KUKA KRL program: ps_ltc_geo_x1.src, ps_ltc_geo_x1.dat

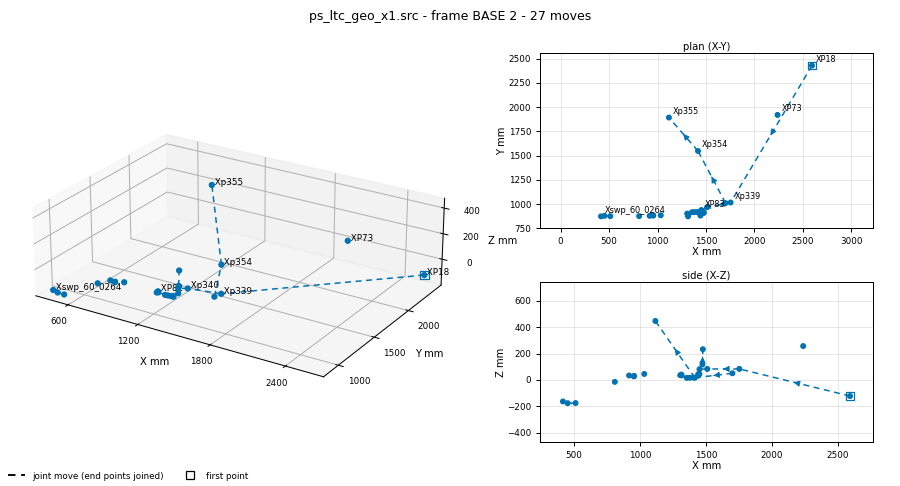
[picture p0: tool path of ps_ltc_geo_x1.src in frame BASE 2, 27 of 45 moves have a stored position in this frame; points joined in program order, loops and branches not executed]
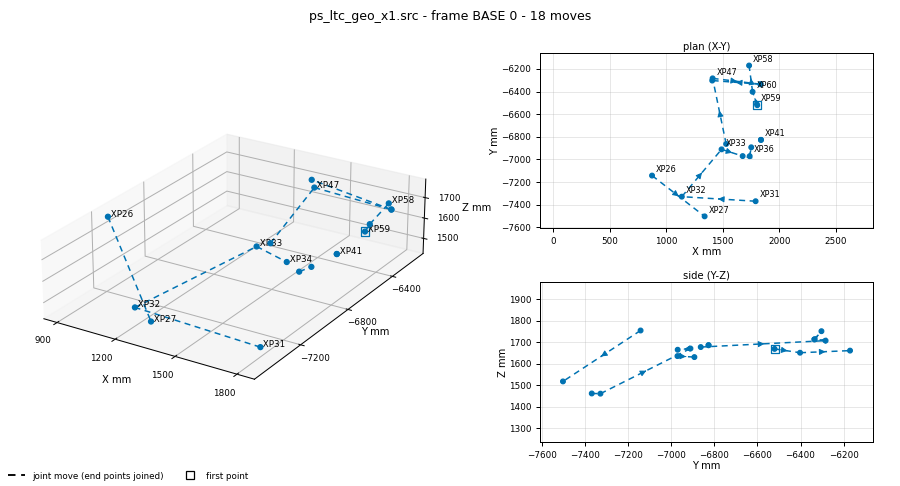
[picture p1: tool path of ps_ltc_geo_x1.src in frame BASE 0, 18 of 45 moves have a stored position in this frame; points joined in program order, loops and branches not executed]
--- ps_ltc_geo_x1.src ---
&ACCESS RVO2
&REL 14
&COMMENT Solda GUN X1 geometria
&PARAM DISKPATH = KRC:\R1\Program\SOLDA LTC
DEF ps_ltc_geo_x1( )

;FOLD INI
  ;FOLD BASISTECH INI
    GLOBAL INTERRUPT DECL 3 WHEN $STOPMESS==TRUE DO IR_STOPM ( )
    INTERRUPT ON 3
    BAS (#INITMOV,0 )
  ;ENDFOLD (BASISTECH INI)
;FOLD SPOTTECH INI
USERSPOT(#INIT)
;ENDFOLD (SPOTTECH INI)
;FOLD GRIPPERTECH INI
USER_GRP(0,DUMMY,DUMMY,GDEFAULT)
;ENDFOLD (GRIPPERTECH INI)
  ;FOLD USER INI
    ;Make your modifications here

  ;ENDFOLD (USER INI)
;ENDFOLD (INI)

; Caracterização dos meios de produção:
; Versão Atual:
; 01/05/2013 12:00 Name: P13.050-R2 CHANGES: Solda Geometria
; Pinça X1, Accelo

chk_w1_wechs_ok ( )    ; CHECK TOOL X1

if MaxStandMenge (4) then
MaxStandmengeErreicht (4)
endif

IF (NOT(GHOST())) THEN
if FraesAnf(4) then
e_fraes1 ()
endif
ENDIF

;FOLD PTP P18 CONT Vel=100 % PDAT100 Tool[1]:Gun X1 Base[2]:Accelo;%{PE}%R 8.2.20,%MKUKATPBASIS,%CMOVE,%VPTP,%P 1:PTP, 2:P18, 3:C_DIS, 5:100, 7:PDAT100
$BWDSTART=FALSE
PDAT_ACT=PPDAT100
FDAT_ACT=FP18
BAS(#PTP_PARAMS,100)
PTP XP18 C_DIS
;ENDFOLD
;FOLD PTP p339 CONT Vel=100 % PDAT30 Tool[1]:Gun X1 Base[2]:Accelo;%{PE}%R 8.2.20,%MKUKATPBASIS,%CMOVE,%VPTP,%P 1:PTP, 2:p339, 3:C_DIS, 5:100, 7:PDAT30
$BWDSTART=FALSE
PDAT_ACT=PPDAT30
FDAT_ACT=Fp339
BAS(#PTP_PARAMS,100)
PTP Xp339 C_DIS
;ENDFOLD
;FOLD PTP p340 CONT Vel=100 % PDAT31 Tool[1]:Gun X1 Base[2]:Accelo;%{PE}%R 8.2.20,%MKUKATPBASIS,%CMOVE,%VPTP,%P 1:PTP, 2:p340, 3:C_DIS, 5:100, 7:PDAT31
$BWDSTART=FALSE
PDAT_ACT=PPDAT31
FDAT_ACT=Fp340
BAS(#PTP_PARAMS,100)
PTP Xp340 C_DIS
;ENDFOLD

;FOLD OUT 3339 'R2 solicita lib. para soldar geometria' State=TRUE ;%{PE}%R 8.2.20,%MKUKATPBASIS,%COUT,%VOUTX,%P 2:3339, 3:R2 solicita lib. para soldar geometria, 5:TRUE, 6:
$OUT[3339]=TRUE
;ENDFOLD
;FOLD WAIT FOR ( IN 3339 'R2 aguarda lib. Soldar geometria' );%{PE}%R 8.2.20,%MKUKATPBASIS,%CEXT_WAIT_FOR,%VEXT_WAIT_FOR,%P 2:, 4:, 5:$IN, 6:3339, 7:R2 aguarda lib.  Soldar geometria, 9:
WAIT FOR  ( $IN[3339] )
;ENDFOLD
;FOLD OUT 3339 'R2 solicita lib. para soldar geometria' State=FALSE ;%{PE}%R 8.2.20,%MKUKATPBASIS,%COUT,%VOUTX,%P 2:3339, 3:R2 solicita lib. para soldar geometria, 5:FALSE, 6:
$OUT[3339]=FALSE
;ENDFOLD
;FOLD OUT 3348 'Fora area GEOBOX' State=FALSE ;%{PE}%R 8.2.20,%MKUKATPBASIS,%COUT,%VOUTX,%P 2:3348, 3:Fora area GEOBOX, 5:FALSE, 6:
$OUT[3348]=FALSE
;ENDFOLD

;FOLD Collision.Monitoring_AREA_1_On ;%{PE}%MKUKATPUSER
COLLSTOP( 7, 1 ) ;not Interrupt-Controlled
;ENDFOLD

;FOLD PTP p341 CONT Vel=100 % PDAT91 Tool[1]:Gun X1 Base[2]:Accelo;%{PE}%R 8.2.20,%MKUKATPBASIS,%CMOVE,%VPTP,%P 1:PTP, 2:p341, 3:C_DIS, 5:100, 7:PDAT91
$BWDSTART=FALSE
PDAT_ACT=PPDAT91
FDAT_ACT=Fp341
BAS(#PTP_PARAMS,100)
PTP Xp341 C_DIS
;ENDFOLD
;FOLD PTP P83 CONT Vel=100 % PDAT166 Tool[1]:Gun X1 Base[2]:Accelo;%{PE}%R 8.2.20,%MKUKATPBASIS,%CMOVE,%VPTP,%P 1:PTP, 2:P83, 3:C_DIS, 5:100, 7:PDAT166
$BWDSTART=FALSE
PDAT_ACT=PPDAT166
FDAT_ACT=FP83
BAS(#PTP_PARAMS,100)
PTP XP83 C_DIS
;ENDFOLD

; SP0328
;FOLD PTP swp_60_0328 PDAT104 SPOT Gun=4 RETR CLS PGNO1=100 ACTIVE=1 Tool[1]:Gun X1 Base[2]:Accelo;%{PE}%R 8.2.2,%MKUKATPSPOT,%CSPOT,%VPTP,%P 1:PTP, 2:swp_60_0328, 3:, 5:100, 7:PDAT104, 10:4, 12:#FIRST, 14:#CLO, 16:181, 18:1, 20:0, 22:0, 24:1, 25:NORMAL
$BWDSTART=FALSE
PDAT_ACT=PPDAT104
FDAT_ACT=Fswp_60_0328
BAS(#PTP_PARAMS,PPDAT104.VEL)
S_ACT.GUN=4
S_ACT.PAIR=SDEFAULT.PAIR
S_ACT.RETR=#CLO
S_ACT.CLO_TM=1
S_ACT.PGNO1=100
S_ACT.PGNO2=SDEFAULT.PGNO2
S_ACT.PRESS1=SDEFAULT.PRESS1
S_ACT.PRESS2=SDEFAULT.PRESS2
S_READY=FALSE
PTP Xswp_60_0328
USERSPOT(#SPOT, S_ACT)
WAIT FOR S_READY
;ENDFOLD

; SP0326
;FOLD PTP swp_60_0326 PDAT157 SPOT Gun=4 RETR OPN PGNO1=132 ACTIVE=1 Tool[1]:Gun X1 Base[2]:Accelo;%{PE}%R 8.2.2,%MKUKATPSPOT,%CSPOT,%VPTP,%P 1:PTP, 2:swp_60_0326, 3:, 5:100, 7:PDAT157, 10:4, 12:#FIRST, 14:#OPN, 16:213, 18:1, 20:0, 22:0, 24:1, 25:NORMAL
$BWDSTART=FALSE
PDAT_ACT=PPDAT157
FDAT_ACT=Fswp_60_0326
BAS(#PTP_PARAMS,PPDAT157.VEL)
S_ACT.GUN=4
S_ACT.PAIR=SDEFAULT.PAIR
S_ACT.RETR=#OPN
S_ACT.CLO_TM=1
S_ACT.PGNO1=132
S_ACT.PGNO2=SDEFAULT.PGNO2
S_ACT.PRESS1=SDEFAULT.PRESS1
S_ACT.PRESS2=SDEFAULT.PRESS2
S_READY=FALSE
PTP Xswp_60_0326
USERSPOT(#SPOT, S_ACT)
WAIT FOR S_READY
;ENDFOLD

; SP0324
;FOLD PTP swp_60_0324 PDAT158 SPOT Gun=4 RETR CLS PGNO1=121 ACTIVE=1 Tool[1]:Gun X1 Base[2]:Accelo;%{PE}%R 8.2.2,%MKUKATPSPOT,%CSPOT,%VPTP,%P 1:PTP, 2:swp_60_0324, 3:, 5:100, 7:PDAT158, 10:4, 12:#FIRST, 14:#CLO, 16:202, 18:1, 20:0, 22:0, 24:1, 25:NORMAL
$BWDSTART=FALSE
PDAT_ACT=PPDAT158
FDAT_ACT=Fswp_60_0324
BAS(#PTP_PARAMS,PPDAT158.VEL)
S_ACT.GUN=4
S_ACT.PAIR=SDEFAULT.PAIR
S_ACT.RETR=#CLO
S_ACT.CLO_TM=1
S_ACT.PGNO1=121
S_ACT.PGNO2=SDEFAULT.PGNO2
S_ACT.PRESS1=SDEFAULT.PRESS1
S_ACT.PRESS2=SDEFAULT.PRESS2
S_READY=FALSE
PTP Xswp_60_0324
USERSPOT(#SPOT, S_ACT)
WAIT FOR S_READY
;ENDFOLD

; SP0322
;FOLD PTP swp_60_0322 PDAT159 SPOT Gun=4 RETR CLS PGNO1=133 ACTIVE=1 Tool[1]:Gun X1 Base[2]:Accelo;%{PE}%R 8.2.2,%MKUKATPSPOT,%CSPOT,%VPTP,%P 1:PTP, 2:swp_60_0322, 3:, 5:100, 7:PDAT159, 10:4, 12:#FIRST, 14:#CLO, 16:214, 18:1, 20:0, 22:0, 24:1, 25:NORMAL
$BWDSTART=FALSE
PDAT_ACT=PPDAT159
FDAT_ACT=Fswp_60_0322
BAS(#PTP_PARAMS,PPDAT159.VEL)
S_ACT.GUN=4
S_ACT.PAIR=SDEFAULT.PAIR
S_ACT.RETR=#CLO
S_ACT.CLO_TM=1
S_ACT.PGNO1=133
S_ACT.PGNO2=SDEFAULT.PGNO2
S_ACT.PRESS1=SDEFAULT.PRESS1
S_ACT.PRESS2=SDEFAULT.PRESS2
S_READY=FALSE
PTP Xswp_60_0322
USERSPOT(#SPOT, S_ACT)
WAIT FOR S_READY
;ENDFOLD

; SP0320
;FOLD PTP swp_60_0320 PDAT160 SPOT Gun=4 RETR OPN PGNO1=134 ACTIVE=1 Tool[1]:Gun X1 Base[2]:Accelo;%{PE}%R 8.2.2,%MKUKATPSPOT,%CSPOT,%VPTP,%P 1:PTP, 2:swp_60_0320, 3:, 5:100, 7:PDAT160, 10:4, 12:#FIRST, 14:#OPN, 16:215, 18:1, 20:0, 22:0, 24:1, 25:NORMAL
$BWDSTART=FALSE
PDAT_ACT=PPDAT160
FDAT_ACT=Fswp_60_0320
BAS(#PTP_PARAMS,PPDAT160.VEL)
S_ACT.GUN=4
S_ACT.PAIR=SDEFAULT.PAIR
S_ACT.RETR=#OPN
S_ACT.CLO_TM=1
S_ACT.PGNO1=134
S_ACT.PGNO2=SDEFAULT.PGNO2
S_ACT.PRESS1=SDEFAULT.PRESS1
S_ACT.PRESS2=SDEFAULT.PRESS2
S_READY=FALSE
PTP Xswp_60_0320
USERSPOT(#SPOT, S_ACT)
WAIT FOR S_READY
;ENDFOLD

; SP0318
;FOLD PTP swp_60_0318 PDAT161 SPOT Gun=4 RETR OPN PGNO1=122 ACTIVE=1 Tool[1]:Gun X1 Base[2]:Accelo;%{PE}%R 8.2.2,%MKUKATPSPOT,%CSPOT,%VPTP,%P 1:PTP, 2:swp_60_0318, 3:, 5:100, 7:PDAT161, 10:4, 12:#FIRST, 14:#OPN, 16:203, 18:1, 20:0, 22:0, 24:1, 25:NORMAL
$BWDSTART=FALSE
PDAT_ACT=PPDAT161
FDAT_ACT=Fswp_60_0318
BAS(#PTP_PARAMS,PPDAT161.VEL)
S_ACT.GUN=4
S_ACT.PAIR=SDEFAULT.PAIR
S_ACT.RETR=#OPN
S_ACT.CLO_TM=1
S_ACT.PGNO1=122
S_ACT.PGNO2=SDEFAULT.PGNO2
S_ACT.PRESS1=SDEFAULT.PRESS1
S_ACT.PRESS2=SDEFAULT.PRESS2
S_READY=FALSE
PTP Xswp_60_0318
USERSPOT(#SPOT, S_ACT)
WAIT FOR S_READY
;ENDFOLD

; SP0316
;FOLD PTP swp_60_0316 PDAT167 SPOT Gun=4 RETR OPN PGNO1=135 ACTIVE=1 Tool[1]:Gun X1 Base[2]:Accelo;%{PE}%R 8.2.2,%MKUKATPSPOT,%CSPOT,%VPTP,%P 1:PTP, 2:swp_60_0316, 3:, 5:100, 7:PDAT167, 10:4, 12:#FIRST, 14:#OPN, 16:216, 18:1, 20:0, 22:0, 24:1, 25:NORMAL
$BWDSTART=FALSE
PDAT_ACT=PPDAT167
FDAT_ACT=Fswp_60_0316
BAS(#PTP_PARAMS,PPDAT167.VEL)
S_ACT.GUN=4
S_ACT.PAIR=SDEFAULT.PAIR
S_ACT.RETR=#OPN
S_ACT.CLO_TM=1
S_ACT.PGNO1=135
S_ACT.PGNO2=SDEFAULT.PGNO2
S_ACT.PRESS1=SDEFAULT.PRESS1
S_ACT.PRESS2=SDEFAULT.PRESS2
S_READY=FALSE
PTP Xswp_60_0316
USERSPOT(#SPOT, S_ACT)
WAIT FOR S_READY
;ENDFOLD

;FOLD PTP P82 CONT Vel=100 % PDAT165 Tool[1]:Gun X1 Base[2]:Accelo;%{PE}%R 8.2.20,%MKUKATPBASIS,%CMOVE,%VPTP,%P 1:PTP, 2:P82, 3:C_DIS, 5:100, 7:PDAT165
$BWDSTART=FALSE
PDAT_ACT=PPDAT165
FDAT_ACT=FP82
BAS(#PTP_PARAMS,100)
PTP XP82 C_DIS
;ENDFOLD
;FOLD PTP P59 CONT Vel=100 % PDAT141 Tool[1]:Gun X1 Base[2]:Accelo;%{PE}%R 8.2.20,%MKUKATPBASIS,%CMOVE,%VPTP,%P 1:PTP, 2:P59, 3:C_DIS, 5:100, 7:PDAT141
$BWDSTART=FALSE
PDAT_ACT=PPDAT141
FDAT_ACT=FP59
BAS(#PTP_PARAMS,100)
PTP XP59 C_DIS
;ENDFOLD
;FOLD PTP P60 CONT Vel=100 % PDAT142 Tool[1]:Gun X1 Base[2]:Accelo;%{PE}%R 8.2.20,%MKUKATPBASIS,%CMOVE,%VPTP,%P 1:PTP, 2:P60, 3:C_DIS, 5:100, 7:PDAT142
$BWDSTART=FALSE
PDAT_ACT=PPDAT142
FDAT_ACT=FP60
BAS(#PTP_PARAMS,100)
PTP XP60 C_DIS
;ENDFOLD
;FOLD PTP P58 CONT Vel=100 % PDAT140 Tool[1]:Gun X1 Base[2]:Accelo;%{PE}%R 8.2.20,%MKUKATPBASIS,%CMOVE,%VPTP,%P 1:PTP, 2:P58, 3:C_DIS, 5:100, 7:PDAT140
$BWDSTART=FALSE
PDAT_ACT=PPDAT140
FDAT_ACT=FP58
BAS(#PTP_PARAMS,100)
PTP XP58 C_DIS
;ENDFOLD
;FOLD PTP P10 Vel=100 % PDAT92 Tool[1]:Gun X1 Base[2]:Accelo;%{PE}%R 8.2.20,%MKUKATPBASIS,%CMOVE,%VPTP,%P 1:PTP, 2:P10, 3:, 5:100, 7:PDAT92
$BWDSTART=FALSE
PDAT_ACT=PPDAT92
FDAT_ACT=FP10
BAS(#PTP_PARAMS,100)
PTP XP10
;ENDFOLD

;FOLD Collision.Monitoring_AREA_1_Off . ;%{PE}%MKUKATPUSER
COLLSTOP( 7, 2+0 )
;ENDFOLD
;FOLD Collision.Monitoring_AREA_2_On ;%{PE}%MKUKATPUSER
COLLSTOP( 8, 1 ) ;not Interrupt-Controlled
;ENDFOLD
;FOLD Collision.Monitoring_4_On ;%{PE}%MKUKATPUSER
COLLSTOP( 4, 1 ) ;Interrupt-Controlled
;ENDFOLD

;FOLD PTP p354 CONT Vel=100 % PDAT44 Tool[1]:Gun X1 Base[2]:Accelo;%{PE}%R 8.2.20,%MKUKATPBASIS,%CMOVE,%VPTP,%P 1:PTP, 2:p354, 3:C_DIS, 5:100, 7:PDAT44
$BWDSTART=FALSE
PDAT_ACT=PPDAT44
FDAT_ACT=Fp354
BAS(#PTP_PARAMS,100)
PTP Xp354 C_DIS
;ENDFOLD
;FOLD PTP p355 CONT Vel=100 % PDAT45 Tool[1]:Gun X1 Base[2]:Accelo;%{PE}%R 8.2.20,%MKUKATPBASIS,%CMOVE,%VPTP,%P 1:PTP, 2:p355, 3:C_DIS, 5:100, 7:PDAT45
$BWDSTART=FALSE
PDAT_ACT=PPDAT45
FDAT_ACT=Fp355
BAS(#PTP_PARAMS,100)
PTP Xp355 C_DIS
;ENDFOLD
;FOLD PTP P26 CONT Vel=100 % PDAT108 Tool[1]:Gun X1 Base[2]:Accelo;%{PE}%R 8.2.20,%MKUKATPBASIS,%CMOVE,%VPTP,%P 1:PTP, 2:P26, 3:C_DIS, 5:100, 7:PDAT108
$BWDSTART=FALSE
PDAT_ACT=PPDAT108
FDAT_ACT=FP26
BAS(#PTP_PARAMS,100)
PTP XP26 C_DIS
;ENDFOLD
;FOLD PTP P27 CONT Vel=100 % PDAT109 Tool[1]:Gun X1 Base[2]:Accelo;%{PE}%R 8.2.20,%MKUKATPBASIS,%CMOVE,%VPTP,%P 1:PTP, 2:P27, 3:C_DIS, 5:100, 7:PDAT109
$BWDSTART=FALSE
PDAT_ACT=PPDAT109
FDAT_ACT=FP27
BAS(#PTP_PARAMS,100)
PTP XP27 C_DIS
;ENDFOLD

; SP0264
;FOLD PTP swp_60_0264 PDAT151 SPOT Gun=4 RETR CLS PGNO1=109 ACTIVE=1 Tool[1]:Gun X1 Base[2]:Accelo;%{PE}%R 8.2.2,%MKUKATPSPOT,%CSPOT,%VPTP,%P 1:PTP, 2:swp_60_0264, 3:, 5:100, 7:PDAT151, 10:4, 12:#FIRST, 14:#CLO, 16:190, 18:1, 20:0, 22:0, 24:1, 25:NORMAL
$BWDSTART=FALSE
PDAT_ACT=PPDAT151
FDAT_ACT=Fswp_60_0264
BAS(#PTP_PARAMS,PPDAT151.VEL)
S_ACT.GUN=4
S_ACT.PAIR=SDEFAULT.PAIR
S_ACT.RETR=#CLO
S_ACT.CLO_TM=1
S_ACT.PGNO1=109
S_ACT.PGNO2=SDEFAULT.PGNO2
S_ACT.PRESS1=SDEFAULT.PRESS1
S_ACT.PRESS2=SDEFAULT.PRESS2
S_READY=FALSE
PTP Xswp_60_0264
USERSPOT(#SPOT, S_ACT)
WAIT FOR S_READY
;ENDFOLD

;FOLD PTP P84 CONT Vel=100 % PDAT168 Tool[1]:Gun X1 Base[2]:Accelo;%{PE}%R 8.2.20,%MKUKATPBASIS,%CMOVE,%VPTP,%P 1:PTP, 2:P84, 3:C_DIS, 5:100, 7:PDAT168
$BWDSTART=FALSE
PDAT_ACT=PPDAT168
FDAT_ACT=FP84
BAS(#PTP_PARAMS,100)
PTP XP84 C_DIS
;ENDFOLD

; SP0268
;FOLD PTP swp_60_0268 PDAT150 SPOT Gun=4 RETR OPN PGNO1=108 ACTIVE=1 Tool[1]:Gun X1 Base[2]:Accelo;%{PE}%R 8.2.2,%MKUKATPSPOT,%CSPOT,%VPTP,%P 1:PTP, 2:swp_60_0268, 3:, 5:100, 7:PDAT150, 10:4, 12:#FIRST, 14:#OPN, 16:189, 18:1, 20:0, 22:0, 24:1, 25:NORMAL
$BWDSTART=FALSE
PDAT_ACT=PPDAT150
FDAT_ACT=Fswp_60_0268
BAS(#PTP_PARAMS,PPDAT150.VEL)
S_ACT.GUN=4
S_ACT.PAIR=SDEFAULT.PAIR
S_ACT.RETR=#OPN
S_ACT.CLO_TM=1
S_ACT.PGNO1=108
S_ACT.PGNO2=SDEFAULT.PGNO2
S_ACT.PRESS1=SDEFAULT.PRESS1
S_ACT.PRESS2=SDEFAULT.PRESS2
S_READY=FALSE
PTP Xswp_60_0268
USERSPOT(#SPOT, S_ACT)
WAIT FOR S_READY
;ENDFOLD

;FOLD PTP P31 CONT Vel=100 % PDAT113 Tool[1]:Gun X1 Base[2]:Accelo;%{PE}%R 8.2.20,%MKUKATPBASIS,%CMOVE,%VPTP,%P 1:PTP, 2:P31, 3:C_DIS, 5:100, 7:PDAT113
$BWDSTART=FALSE
PDAT_ACT=PPDAT113
FDAT_ACT=FP31
BAS(#PTP_PARAMS,100)
PTP XP31 C_DIS
;ENDFOLD
;FOLD PTP P32 CONT Vel=100 % PDAT114 Tool[1]:Gun X1 Base[2]:Accelo;%{PE}%R 8.2.20,%MKUKATPBASIS,%CMOVE,%VPTP,%P 1:PTP, 2:P32, 3:C_DIS, 5:100, 7:PDAT114
$BWDSTART=FALSE
PDAT_ACT=PPDAT114
FDAT_ACT=FP32
BAS(#PTP_PARAMS,100)
PTP XP32 C_DIS
;ENDFOLD
;FOLD PTP P33 CONT Vel=100 % PDAT115 Tool[1]:Gun X1 Base[2]:Accelo;%{PE}%R 8.2.20,%MKUKATPBASIS,%CMOVE,%VPTP,%P 1:PTP, 2:P33, 3:C_DIS, 5:100, 7:PDAT115
$BWDSTART=FALSE
PDAT_ACT=PPDAT115
FDAT_ACT=FP33
BAS(#PTP_PARAMS,100)
PTP XP33 C_DIS
;ENDFOLD
;FOLD PTP P34 CONT Vel=100 % PDAT116 Tool[1]:Gun X1 Base[2]:Accelo;%{PE}%R 8.2.20,%MKUKATPBASIS,%CMOVE,%VPTP,%P 1:PTP, 2:P34, 3:C_DIS, 5:100, 7:PDAT116
$BWDSTART=FALSE
PDAT_ACT=PPDAT116
FDAT_ACT=FP34
BAS(#PTP_PARAMS,100)
PTP XP34 C_DIS
;ENDFOLD

; SP0284
;FOLD PTP swp_60_0284 PDAT143 SPOT Gun=4 RETR OPN PGNO1=107 ACTIVE=1 Tool[1]:Gun X1 Base[2]:Accelo;%{PE}%R 8.2.2,%MKUKATPSPOT,%CSPOT,%VPTP,%P 1:PTP, 2:swp_60_0284, 3:, 5:100, 7:PDAT143, 10:4, 12:#FIRST, 14:#OPN, 16:188, 18:1, 20:0, 22:0, 24:1, 25:NORMAL
$BWDSTART=FALSE
PDAT_ACT=PPDAT143
FDAT_ACT=Fswp_60_0284
BAS(#PTP_PARAMS,PPDAT143.VEL)
S_ACT.GUN=4
S_ACT.PAIR=SDEFAULT.PAIR
S_ACT.RETR=#OPN
S_ACT.CLO_TM=1
S_ACT.PGNO1=107
S_ACT.PGNO2=SDEFAULT.PGNO2
S_ACT.PRESS1=SDEFAULT.PRESS1
S_ACT.PRESS2=SDEFAULT.PRESS2
S_READY=FALSE
PTP Xswp_60_0284
USERSPOT(#SPOT, S_ACT)
WAIT FOR S_READY
;ENDFOLD

;FOLD PTP P36 CONT Vel=100 % PDAT118 Tool[1]:Gun X1 Base[2]:Accelo;%{PE}%R 8.2.20,%MKUKATPBASIS,%CMOVE,%VPTP,%P 1:PTP, 2:P36, 3:C_DIS, 5:100, 7:PDAT118
$BWDSTART=FALSE
PDAT_ACT=PPDAT118
FDAT_ACT=FP36
BAS(#PTP_PARAMS,100)
PTP XP36 C_DIS
;ENDFOLD
;FOLD PTP P37 CONT Vel=100 % PDAT119 Tool[1]:Gun X1 Base[2]:Accelo;%{PE}%R 8.2.20,%MKUKATPBASIS,%CMOVE,%VPTP,%P 1:PTP, 2:P37, 3:C_DIS, 5:100, 7:PDAT119
$BWDSTART=FALSE
PDAT_ACT=PPDAT119
FDAT_ACT=FP37
BAS(#PTP_PARAMS,100)
PTP XP37 C_DIS
;ENDFOLD
;FOLD PTP P62 PDAT144 RETR CLS Gun=4 Tool[1]:Gun X1 Base[2]:Accelo;%{PE}%R 8.2.2,%MKUKATPSPOT,%CRETR,%VPTP,%P 1:PTP, 2:P62, 3:, 5:100, 7:PDAT144, 9:#CLO, 11:4, 13:#FIRST
$BWDSTART=FALSE
PDAT_ACT=PPDAT144
FDAT_ACT=FP62
BAS(#PTP_PARAMS,PPDAT144.VEL)
S_ACT.GUN=4
S_ACT.PAIR=#FIRST
S_ACT.RETR=#CLO
S_READY=FALSE
PTP XP62
USERSPOT(#RETR, S_ACT)
WAIT FOR S_READY
;ENDFOLD

; SP0290
;FOLD PTP swp_60_0290 PDAT145 SPOT Gun=4 RETR CLS PGNO1=106 ACTIVE=1 Tool[1]:Gun X1 Base[2]:Accelo;%{PE}%R 8.2.2,%MKUKATPSPOT,%CSPOT,%VPTP,%P 1:PTP, 2:swp_60_0290, 3:, 5:100, 7:PDAT145, 10:4, 12:#FIRST, 14:#CLO, 16:187, 18:1, 20:0, 22:0, 24:1, 25:NORMAL
$BWDSTART=FALSE
PDAT_ACT=PPDAT145
FDAT_ACT=Fswp_60_0290
BAS(#PTP_PARAMS,PPDAT145.VEL)
S_ACT.GUN=4
S_ACT.PAIR=SDEFAULT.PAIR
S_ACT.RETR=#CLO
S_ACT.CLO_TM=1
S_ACT.PGNO1=106
S_ACT.PGNO2=SDEFAULT.PGNO2
S_ACT.PRESS1=SDEFAULT.PRESS1
S_ACT.PRESS2=SDEFAULT.PRESS2
S_READY=FALSE
PTP Xswp_60_0290
USERSPOT(#SPOT, S_ACT)
WAIT FOR S_READY
;ENDFOLD

;FOLD PTP P41 CONT Vel=100 % PDAT123 Tool[1]:Gun X1 Base[2]:Accelo;%{PE}%R 8.2.20,%MKUKATPBASIS,%CMOVE,%VPTP,%P 1:PTP, 2:P41, 3:C_DIS, 5:100, 7:PDAT123
$BWDSTART=FALSE
PDAT_ACT=PPDAT123
FDAT_ACT=FP41
BAS(#PTP_PARAMS,100)
PTP XP41 C_DIS
;ENDFOLD

; SP0296
;FOLD PTP swp_60_0296 PDAT147 SPOT Gun=4 RETR CLS PGNO1=105 ACTIVE=1 Tool[1]:Gun X1 Base[2]:Accelo;%{PE}%R 8.2.2,%MKUKATPSPOT,%CSPOT,%VPTP,%P 1:PTP, 2:swp_60_0296, 3:, 5:100, 7:PDAT147, 10:4, 12:#FIRST, 14:#CLO, 16:186, 18:1, 20:0, 22:0, 24:1, 25:NORMAL
$BWDSTART=FALSE
PDAT_ACT=PPDAT147
FDAT_ACT=Fswp_60_0296
BAS(#PTP_PARAMS,PPDAT147.VEL)
S_ACT.GUN=4
S_ACT.PAIR=SDEFAULT.PAIR
S_ACT.RETR=#CLO
S_ACT.CLO_TM=1
S_ACT.PGNO1=105
S_ACT.PGNO2=SDEFAULT.PGNO2
S_ACT.PRESS1=SDEFAULT.PRESS1
S_ACT.PRESS2=SDEFAULT.PRESS2
S_READY=FALSE
PTP Xswp_60_0296
USERSPOT(#SPOT, S_ACT)
WAIT FOR S_READY
;ENDFOLD

;FOLD Collision.Monitoring_AREA_2_Off . ;%{PE}%MKUKATPUSER
COLLSTOP( 8, 2+0 )
;ENDFOLD
;FOLD Collision.Monitoring_AREA_3_On ;%{PE}%MKUKATPUSER
COLLSTOP( 9, 1 ) ;not Interrupt-Controlled
;ENDFOLD

;FOLD PTP P43 CONT Vel=100 % PDAT125 Tool[1]:Gun X1 Base[2]:Accelo;%{PE}%R 8.2.20,%MKUKATPBASIS,%CMOVE,%VPTP,%P 1:PTP, 2:P43, 3:C_DIS, 5:100, 7:PDAT125
$BWDSTART=FALSE
PDAT_ACT=PPDAT125
FDAT_ACT=FP43
BAS(#PTP_PARAMS,100)
PTP XP43 C_DIS
;ENDFOLD
;FOLD PTP P71 PDAT153 RETR OPN Gun=4 Tool[1]:Gun X1 Base[2]:Accelo;%{PE}%R 8.2.2,%MKUKATPSPOT,%CRETR,%VPTP,%P 1:PTP, 2:P71, 3:, 5:100, 7:PDAT153, 9:#OPN, 11:4, 13:#FIRST
$BWDSTART=FALSE
PDAT_ACT=PPDAT153
FDAT_ACT=FP71
BAS(#PTP_PARAMS,PPDAT153.VEL)
S_ACT.GUN=4
S_ACT.PAIR=#FIRST
S_ACT.RETR=#OPN
S_READY=FALSE
PTP XP71
USERSPOT(#RETR, S_ACT)
WAIT FOR S_READY
;ENDFOLD
;FOLD PTP P45 CONT Vel=100 % PDAT127 Tool[1]:Gun X1 Base[2]:Accelo;%{PE}%R 8.2.20,%MKUKATPBASIS,%CMOVE,%VPTP,%P 1:PTP, 2:P45, 3:C_DIS, 5:100, 7:PDAT127
$BWDSTART=FALSE
PDAT_ACT=PPDAT127
FDAT_ACT=FP45
BAS(#PTP_PARAMS,100)
PTP XP45 C_DIS
;ENDFOLD
;FOLD PTP P47 CONT Vel=100 % PDAT129 Tool[1]:Gun X1 Base[2]:Accelo;%{PE}%R 8.2.20,%MKUKATPBASIS,%CMOVE,%VPTP,%P 1:PTP, 2:P47, 3:C_DIS, 5:100, 7:PDAT129
$BWDSTART=FALSE
PDAT_ACT=PPDAT129
FDAT_ACT=FP47
BAS(#PTP_PARAMS,100)
PTP XP47 C_DIS
;ENDFOLD
;FOLD PTP P48 CONT Vel=100 % PDAT130 Tool[1]:Gun X1 Base[2]:Accelo;%{PE}%R 8.2.20,%MKUKATPBASIS,%CMOVE,%VPTP,%P 1:PTP, 2:P48, 3:C_DIS, 5:100, 7:PDAT130
$BWDSTART=FALSE
PDAT_ACT=PPDAT130
FDAT_ACT=FP48
BAS(#PTP_PARAMS,100)
PTP XP48 C_DIS
;ENDFOLD

; SP0350
;FOLD PTP swp_60_0350 PDAT148 SPOT Gun=4 RETR CLS PGNO1=104 ACTIVE=1 Tool[1]:Gun X1 Base[2]:Accelo;%{PE}%R 8.2.2,%MKUKATPSPOT,%CSPOT,%VPTP,%P 1:PTP, 2:swp_60_0350, 3:, 5:100, 7:PDAT148, 10:4, 12:#FIRST, 14:#CLO, 16:185, 18:1, 20:0, 22:0, 24:1, 25:NORMAL
$BWDSTART=FALSE
PDAT_ACT=PPDAT148
FDAT_ACT=Fswp_60_0350
BAS(#PTP_PARAMS,PPDAT148.VEL)
S_ACT.GUN=4
S_ACT.PAIR=SDEFAULT.PAIR
S_ACT.RETR=#CLO
S_ACT.CLO_TM=1
S_ACT.PGNO1=104
S_ACT.PGNO2=SDEFAULT.PGNO2
S_ACT.PRESS1=SDEFAULT.PRESS1
S_ACT.PRESS2=SDEFAULT.PRESS2
S_READY=FALSE
PTP Xswp_60_0350
USERSPOT(#SPOT, S_ACT)
WAIT FOR S_READY
;ENDFOLD

; SP0356
;FOLD PTP swp_60_0356 PDAT149 SPOT Gun=4 RETR OPN PGNO1=103 ACTIVE=1 Tool[1]:Gun X1 Base[2]:Accelo;%{PE}%R 8.2.2,%MKUKATPSPOT,%CSPOT,%VPTP,%P 1:PTP, 2:swp_60_0356, 3:, 5:100, 7:PDAT149, 10:4, 12:#FIRST, 14:#OPN, 16:184, 18:1, 20:0, 22:0, 24:1, 25:NORMAL
$BWDSTART=FALSE
PDAT_ACT=PPDAT149
FDAT_ACT=Fswp_60_0356
BAS(#PTP_PARAMS,PPDAT149.VEL)
S_ACT.GUN=4
S_ACT.PAIR=SDEFAULT.PAIR
S_ACT.RETR=#OPN
S_ACT.CLO_TM=1
S_ACT.PGNO1=103
S_ACT.PGNO2=SDEFAULT.PGNO2
S_ACT.PRESS1=SDEFAULT.PRESS1
S_ACT.PRESS2=SDEFAULT.PRESS2
S_READY=FALSE
PTP Xswp_60_0356
USERSPOT(#SPOT, S_ACT)
WAIT FOR S_READY
;ENDFOLD

;FOLD PTP P52 CONT Vel=100 % PDAT134 Tool[1]:Gun X1 Base[2]:Accelo;%{PE}%R 8.2.20,%MKUKATPBASIS,%CMOVE,%VPTP,%P 1:PTP, 2:P52, 3:C_DIS, 5:100, 7:PDAT134
$BWDSTART=FALSE
PDAT_ACT=PPDAT134
FDAT_ACT=FP52
BAS(#PTP_PARAMS,100)
PTP XP52 C_DIS
;ENDFOLD
;FOLD PTP P53 CONT Vel=100 % PDAT135 Tool[1]:Gun X1 Base[2]:Accelo;%{PE}%R 8.2.20,%MKUKATPBASIS,%CMOVE,%VPTP,%P 1:PTP, 2:P53, 3:C_DIS, 5:100, 7:PDAT135
$BWDSTART=FALSE
PDAT_ACT=PPDAT135
FDAT_ACT=FP53
BAS(#PTP_PARAMS,100)
PTP XP53 C_DIS
;ENDFOLD
;FOLD PTP P73 Vel=100 % PDAT155 Tool[1]:Gun X1 Base[2]:Accelo;%{PE}%R 8.2.20,%MKUKATPBASIS,%CMOVE,%VPTP,%P 1:PTP, 2:P73, 3:, 5:100, 7:PDAT155
$BWDSTART=FALSE
PDAT_ACT=PPDAT155
FDAT_ACT=FP73
BAS(#PTP_PARAMS,100)
PTP XP73
;ENDFOLD

;FOLD Collision.Monitoring_4_Off . ;%{PE}%MKUKATPUSER
COLLSTOP( 4, 2+0 )
;ENDFOLD
;FOLD Collision.Monitoring_AREA_3_Off . ;%{PE}%MKUKATPUSER
COLLSTOP( 9, 2+0 )
;ENDFOLD

;FOLD OUT 3348 'Fora area GEOBOX' State=TRUE ;%{PE}%R 8.2.20,%MKUKATPBASIS,%COUT,%VOUTX,%P 2:3348, 3:Fora area GEOBOX, 5:TRUE, 6:
$OUT[3348]=TRUE
;ENDFOLD

IF (NOT(GHOST())) THEN
if FraesAnf(4) then
f_fraes1 ()
endif
ENDIF

END

--- ps_ltc_geo_x1.dat ---
&ACCESS RVO2
&REL 14
&COMMENT Solda GUN X1 geometria
&PARAM DISKPATH = KRC:\R1\Program\SOLDA LTC
DEFDAT  ps_ltc_geo_x1
;FOLD EXTERNAL DECLARATIONS;%{PE}%MKUKATPBASIS,%CEXT,%VCOMMON,%P
;FOLD GRIPPERTECH EXT
EXT  H50 (INT  :IN,INT  :IN,INT  :IN,GRP_TYP  :IN )
;ENDFOLD (GRIPPERTECH EXT)
;FOLD SPOTTECH EXT
EXT  USERSPOT (S_COMMAND  :IN,SPOT_TYPE  :IN )
;ENDFOLD (SPOTTECH EXT)
;FOLD BASISTECH EXT;%{PE}%MKUKATPBASIS,%CEXT,%VEXT,%P
EXT  BAS (BAS_COMMAND  :IN,REAL  :IN )
DECL INT SUCCESS
;ENDFOLD (BASISTECH EXT)
;FOLD USER EXT;%{E}%MKUKATPUSER,%CEXT,%VEXT,%P
;Make your modifications here

;ENDFOLD (USER EXT)
;ENDFOLD (EXTERNAL DECLARATIONS)

;# ============ START PATH : swp_p13050r2_ltc_geo_x1 =============
DECL FDAT Fswp_60_0326={TOOL_NO 1,BASE_NO 2,IPO_FRAME #BASE,POINT2[] " ",TQ_STATE FALSE}
DECL SPOT_TYPE SS_OLP1={GUN 1,PAIR #FIRST,RETR #OPN,CLO_TM 0,PGNO1 1,PRESS1 1.0,PGNO2 0,PRESS2 0.0}
DECL E6POS Xswp_60_0326={X 1440.89099,Y 894.045471,Z 31.5168095,A -159.997894,B -3.0173409,C -140.140106,S 2,T 35,E1 -4617.46387,E2 0.0,E3 0.0,E4 0.0,E5 0.0,E6 0.0}
DECL FDAT Fswp_60_0322={TOOL_NO 1,BASE_NO 2,IPO_FRAME #BASE,POINT2[] " "}
DECL SPOT_TYPE SS_OLP2={GUN 1,PAIR #FIRST,RETR #OPN,CLO_TM 0,PGNO1 1,PRESS1 1.0,PGNO2 0,PRESS2 0.0}
DECL E6POS Xswp_60_0322={X 1379.50696,Y 917.822388,Z 16.3037205,A -171.276505,B -1.12520099,C -145.708496,S 2,T 35,E1 -4617.46094,E2 0.0,E3 0.0,E4 0.0,E5 0.0,E6 0.0}
DECL FDAT Fswp_60_0318={TOOL_NO 1,BASE_NO 2,IPO_FRAME #BASE,POINT2[] " "}
DECL SPOT_TYPE SS_OLP3={GUN 1,PAIR #FIRST,RETR #OPN,CLO_TM 0,PGNO1 1,PRESS1 1.0,PGNO2 0,PRESS2 0.0}
DECL E6POS Xswp_60_0318={X 1316.23206,Y 893.451721,Z 34.1688995,A -171.866196,B -2.02005601,C -146.172501,S 2,T 35,E1 -4617.52979,E2 0.0,E3 0.0,E4 0.0,E5 0.0,E6 0.0}
DECL FDAT Fswp_60_0356={TOOL_NO 1,BASE_NO 2,IPO_FRAME #BASE,POINT2[] " "}
DECL SPOT_TYPE SS_OLP4={GUN 1,PAIR #FIRST,RETR #OPN,CLO_TM 0,PGNO1 1,PRESS1 1.0,PGNO2 0,PRESS2 0.0}
DECL E6POS Xswp_60_0356={X 1477.68201,Y 913.010681,Z 232.539505,A -91.0726166,B -4.99526501,C 89.5052872,S 6,T 51,E1 -4829.7959,E2 0.0,E3 0.0,E4 0.0,E5 0.0,E6 0.0}
DECL FDAT Fswp_60_0350={TOOL_NO 1,BASE_NO 2,IPO_FRAME #BASE,POINT2[] " "}
DECL SPOT_TYPE SS_OLP5={GUN 1,PAIR #FIRST,RETR #OPN,CLO_TM 0,PGNO1 1,PRESS1 1.0,PGNO2 0,PRESS2 0.0}
DECL E6POS Xswp_60_0350={X 1474.26501,Y 909.548706,Z 116.354202,A -91.1325912,B 4.90854406,C 89.584198,S 6,T 51,E1 -4829.7959,E2 0.0,E3 0.0,E4 0.0,E5 0.0,E6 0.0}
DECL FDAT Fswp_60_0296={TOOL_NO 1,BASE_NO 2,IPO_FRAME #BASE,POINT2[] " "}
DECL SPOT_TYPE SS_OLP6={GUN 1,PAIR #FIRST,RETR #OPN,CLO_TM 0,PGNO1 1,PRESS1 1.0,PGNO2 0,PRESS2 0.0}
DECL E6POS Xswp_60_0296={X 1033.53198,Y 884.917114,Z 45.0556412,A -90.2147217,B 19.7881393,C 15.1591501,S 6,T 19,E1 -4845.0249,E2 0.0,E3 0.0,E4 0.0,E5 0.0,E6 0.0}
DECL FDAT Fswp_60_0290={TOOL_NO 1,BASE_NO 2,IPO_FRAME #BASE,POINT2[] " "}
DECL SPOT_TYPE SS_OLP7={GUN 1,PAIR #FIRST,RETR #OPN,CLO_TM 0,PGNO1 1,PRESS1 1.0,PGNO2 0,PRESS2 0.0}
DECL E6POS Xswp_60_0290={X 918.688782,Y 879.437805,Z 33.3725395,A -96.8630524,B 14.4618196,C 10.1200705,S 6,T 19,E1 -4845.01807,E2 0.0,E3 0.0,E4 0.0,E5 0.0,E6 0.0}
DECL FDAT Fswp_60_0284={TOOL_NO 1,BASE_NO 2,IPO_FRAME #BASE,POINT2[] " "}
DECL SPOT_TYPE SS_OLP8={GUN 1,PAIR #FIRST,RETR #OPN,CLO_TM 0,PGNO1 1,PRESS1 1.0,PGNO2 0,PRESS2 0.0}
DECL E6POS Xswp_60_0284={X 810.263184,Y 876.497681,Z -14.9003096,A -101.040604,B 20.5212498,C 26.0307407,S 6,T 19,E1 -4845.02393,E2 0.0,E3 0.0,E4 0.0,E5 0.0,E6 0.0}
DECL FDAT Fswp_60_0268={TOOL_NO 1,BASE_NO 2,IPO_FRAME #BASE,POINT2[] " "}
DECL SPOT_TYPE SS_OLP9={GUN 1,PAIR #FIRST,RETR #OPN,CLO_TM 0,PGNO1 1,PRESS1 1.0,PGNO2 0,PRESS2 0.0}
DECL E6POS Xswp_60_0268={X 512.70282,Y 875.895813,Z -175.678207,A -80.5816193,B 5.79682779,C 5.26112223,S 6,T 19,E1 -5459.71387,E2 0.0,E3 0.0,E4 0.0,E5 0.0,E6 0.0}
DECL FDAT Fswp_60_0264={TOOL_NO 1,BASE_NO 2,IPO_FRAME #BASE,POINT2[] " "}
DECL SPOT_TYPE SS_OLP10={GUN 1,PAIR #FIRST,RETR #OPN,CLO_TM 0,PGNO1 1,PRESS1 1.0,PGNO2 0,PRESS2 0.0}
DECL E6POS Xswp_60_0264={X 417.230286,Y 874.02771,Z -163.492096,A -83.0655136,B 11.3301601,C -19.7582703,S 6,T 19,E1 -5459.74023,E2 0.0,E3 0.0,E4 0.0,E5 0.0,E6 0.0}
DECL BASIS_SUGG_T LAST_BASIS={POINT1[] "P84                     ",POINT2[] "P84                     ",CP_PARAMS[] "CPDAT0                  ",PTP_PARAMS[] "PDAT168                 ",CONT[] "C_DIS                   ",CP_VEL[] "2.0                     ",PTP_VEL[] "100                     ",SPL_NAME[] "S0                      "}
DECL SPOT_SUGG_T LAST_SPOT={GUN[] "4                       ",RETR_CMD[] "#OPN                    ",CHOISE[] "#FIRST                  ",CLO_TM[] "1                       ",PGNO1[] "203                     ",PRESS1[] "0                       ",PGNO2[] "1                       ",PRESS2[] "0                       ",SPOT_PARAMS[] "NORMAL                  "}
DECL E6POS XP339={X 1754.13196,Y 1016.74298,Z 83.1492615,A -164.185501,B 18.5443897,C -158.434204,S 2,T 35,E1 -4458.23779,E2 0.0,E3 0.0,E4 0.0,E5 0.0,E6 0.0}
DECL FDAT Fp339={TOOL_NO 1,BASE_NO 2,IPO_FRAME #BASE,POINT2[] " ",TQ_STATE FALSE}
DECL PDAT PPDAT30={VEL 100.0,ACC 100.0,APO_DIST 100.0,APO_MODE #CDIS}
DECL E6POS XP340={X 1511.08801,Y 967.887085,Z 82.8026428,A -169.680405,B 7.87629414,C -159.822693,S 2,T 35,E1 -4617.45313,E2 0.0,E3 0.0,E4 0.0,E5 0.0,E6 0.0}
DECL FDAT Fp340={TOOL_NO 1,BASE_NO 2,IPO_FRAME #BASE,POINT2[] " ",TQ_STATE FALSE}
DECL PDAT PPDAT31={VEL 100.0,ACC 100.0,APO_DIST 100.0,APO_MODE #CDIS}
DECL E6POS XP341={X 1451.83398,Y 937.507507,Z 81.1336823,A -171.963394,B 1.64496303,C -160.012405,S 2,T 35,E1 -4617.45313,E2 0.0,E3 0.0,E4 0.0,E5 0.0,E6 0.0}
DECL FDAT Fp341={TOOL_NO 1,BASE_NO 2,IPO_FRAME #BASE,POINT2[] " ",TQ_STATE FALSE}
DECL E6POS XP354={X 1417.54895,Y 1548.25305,Z 16.3868809,A -170.275406,B 20.6585407,C -155.272598,S 2,T 35,E1 -4617.31299,E2 0.0,E3 0.0,E4 0.0,E5 0.0,E6 0.0}
DECL FDAT Fp354={TOOL_NO 1,BASE_NO 2,IPO_FRAME #BASE,POINT2[] " ",TQ_STATE FALSE}
DECL PDAT PPDAT44={VEL 100.0,ACC 100.0,APO_DIST 100.0,APO_MODE #CDIS}
DECL E6POS XP355={X 1117.578,Y 1893.255,Z 446.7435,A -149.1931,B 7.65658712,C -137.427094,S 6,T 51,E1 -4617.31299,E2 0.0,E3 0.0,E4 0.0,E5 0.0,E6 0.0}
DECL FDAT Fp355={TOOL_NO 1,BASE_NO 2,IPO_FRAME #BASE,POINT2[] " ",TQ_STATE FALSE}
DECL PDAT PPDAT45={VEL 100.0,ACC 100.0,APO_DIST 100.0,APO_MODE #CDIS}
DECL PDAT PPDAT91={VEL 100.0,ACC 100.0,APO_DIST 20.0,APO_MODE #CDIS}
DECL PDAT PPDAT92={VEL 100.0,ACC 100.0,APO_DIST 100.0,APO_MODE #CDIS}
DECL E6POS XP10={X 1701.64502,Y 1010.94202,Z 50.3210602,A -171.141296,B 15.6092701,C -169.974899,S 2,T 35,E1 -4617.31299,E2 0.0,E3 0.0,E4 0.0,E5 0.0,E6 0.0}
DECL FDAT FP10={TOOL_NO 1,BASE_NO 2,IPO_FRAME #BASE,POINT2[] " ",TQ_STATE FALSE}
DECL PDAT PPDAT100={VEL 100.0,ACC 100.0,APO_DIST 100.0,APO_MODE #CDIS}
DECL E6POS XP18={X 2593.28198,Y 2429.84009,Z -122.263496,A -172.544495,B 61.4785881,C 178.740707,S 2,T 35,E1 -3217.95093,E2 0.0,E3 0.0,E4 0.0,E5 0.0,E6 0.0}
DECL FDAT FP18={TOOL_NO 1,BASE_NO 2,IPO_FRAME #BASE,POINT2[] " ",TQ_STATE FALSE}
DECL PDAT PPDAT104={VEL 100.0,ACC 100.0,APO_DIST 100.0,APO_MODE #CDIS}
DECL E6POS XP26={X 875.52887,Y -7142.63721,Z 1754.10303,A -42.8865509,B 20.2833996,C 87.7021866,S 6,T 50,E1 -4807.50391,E2 0.0,E3 0.0,E4 0.0,E5 0.0,E6 0.0}
DECL FDAT FP26={TOOL_NO 1,BASE_NO 0,IPO_FRAME #BASE,POINT2[] " ",TQ_STATE FALSE}
DECL PDAT PPDAT108={VEL 100.0,ACC 100.0,APO_DIST 100.0,APO_MODE #CDIS}
DECL E6POS XP27={X 1340.20398,Y -7503.00586,Z 1517.61804,A -19.7759609,B 19.0676498,C -7.15892315,S 6,T 18,E1 -5125.43994,E2 0.0,E3 0.0,E4 0.0,E5 0.0,E6 0.0}
DECL FDAT FP27={TOOL_NO 1,BASE_NO 0,IPO_FRAME #BASE,POINT2[] " ",TQ_STATE FALSE}
DECL PDAT PPDAT109={VEL 100.0,ACC 100.0,APO_DIST 100.0,APO_MODE #CDIS}
DECL E6POS XP31={X 1790.88599,Y -7369.36914,Z 1461.67297,A 3.54338598,B 6.05099392,C 5.29669189,S 6,T 19,E1 -5459.73877,E2 0.0,E3 0.0,E4 0.0,E5 0.0,E6 0.0}
DECL FDAT FP31={TOOL_NO 1,BASE_NO 0,IPO_FRAME #BASE,POINT2[] " ",TQ_STATE FALSE}
DECL PDAT PPDAT113={VEL 100.0,ACC 100.0,APO_DIST 100.0,APO_MODE #CDIS}
DECL E6POS XP32={X 1138.55005,Y -7329.03516,Z 1460.82703,A -24.8452702,B 10.6812496,C 4.63611889,S 6,T 18,E1 -4941.47217,E2 0.0,E3 0.0,E4 0.0,E5 0.0,E6 0.0}
DECL FDAT FP32={TOOL_NO 1,BASE_NO 0,IPO_FRAME #BASE,POINT2[] " ",TQ_STATE FALSE}
DECL PDAT PPDAT114={VEL 100.0,ACC 100.0,APO_DIST 100.0,APO_MODE #CDIS}
DECL E6POS XP33={X 1489.85596,Y -6911.00586,Z 1670.39795,A -11.8927603,B 15.9203901,C 14.7493296,S 6,T 19,E1 -4941.48291,E2 0.0,E3 0.0,E4 0.0,E5 0.0,E6 0.0}
DECL FDAT FP33={TOOL_NO 1,BASE_NO 0,IPO_FRAME #BASE,POINT2[] " ",TQ_STATE FALSE}
DECL PDAT PPDAT115={VEL 100.0,ACC 100.0,APO_DIST 100.0,APO_MODE #CDIS}
DECL E6POS XP34={X 1676.35901,Y -6970.3291,Z 1664.69702,A -10.8957005,B 19.3892708,C 26.3331509,S 6,T 19,E1 -4845.02588,E2 0.0,E3 0.0,E4 0.0,E5 0.0,E6 0.0}
DECL FDAT FP34={TOOL_NO 1,BASE_NO 0,IPO_FRAME #BASE,POINT2[] " ",TQ_STATE FALSE}
DECL PDAT PPDAT116={VEL 100.0,ACC 100.0,APO_DIST 100.0,APO_MODE #CDIS}
DECL E6POS XP36={X 1738.40601,Y -6971.35596,Z 1635.21301,A -11.03932,B 20.5207005,C 26.0304108,S 6,T 19,E1 -4845.02588,E2 0.0,E3 0.0,E4 0.0,E5 0.0,E6 0.0}
DECL FDAT FP36={TOOL_NO 1,BASE_NO 0,IPO_FRAME #BASE,POINT2[] " ",TQ_STATE FALSE}
DECL PDAT PPDAT118={VEL 100.0,ACC 100.0,APO_DIST 100.0,APO_MODE #CDIS}
DECL E6POS XP37={X 1752.21899,Y -6892.74805,Z 1630.56995,A -11.04037,B 20.5200901,C 10.7065401,S 6,T 19,E1 -4845.02686,E2 0.0,E3 0.0,E4 0.0,E5 0.0,E6 0.0}
DECL FDAT FP37={TOOL_NO 1,BASE_NO 0,IPO_FRAME #BASE,POINT2[] " ",TQ_STATE FALSE}
DECL PDAT PPDAT119={VEL 100.0,ACC 100.0,APO_DIST 100.0,APO_MODE #CDIS}
DECL E6POS XP41={X 1838.07397,Y -6827.02783,Z 1685.75098,A -3.05619192,B 18.9826794,C 6.31875801,S 6,T 19,E1 -4845.01904,E2 0.0,E3 0.0,E4 0.0,E5 0.0,E6 0.0}
DECL FDAT FP41={TOOL_NO 1,BASE_NO 0,IPO_FRAME #BASE,POINT2[] " ",TQ_STATE FALSE}
DECL PDAT PPDAT123={VEL 100.0,ACC 100.0,APO_DIST 100.0,APO_MODE #CDIS}
DECL E6POS XP43={X 1838.07397,Y -6827.02783,Z 1685.75098,A -3.05619097,B 18.9826794,C 6.31875706,S 6,T 19,E1 -4845.02002,E2 0.0,E3 0.0,E4 0.0,E5 0.0,E6 0.0}
DECL FDAT FP43={TOOL_NO 1,BASE_NO 0,IPO_FRAME #BASE,POINT2[] " ",TQ_STATE FALSE}
DECL PDAT PPDAT125={VEL 100.0,ACC 100.0,APO_DIST 100.0,APO_MODE #CDIS}
DECL E6POS XP45={X 1530.41699,Y -6863.25391,Z 1677.14697,A -8.84182453,B 14.9026804,C 12.4745197,S 6,T 19,E1 -4803.97803,E2 0.0,E3 0.0,E4 0.0,E5 0.0,E6 0.0}
DECL FDAT FP45={TOOL_NO 1,BASE_NO 0,IPO_FRAME #BASE,POINT2[] " ",TQ_STATE FALSE}
DECL PDAT PPDAT127={VEL 100.0,ACC 100.0,APO_DIST 100.0,APO_MODE #CDIS}
DECL E6POS XP47={X 1410.80005,Y -6283.52197,Z 1706.96106,A 0.0430345498,B 9.15813065,C 88.8373337,S 6,T 50,E1 -4829.79492,E2 0.0,E3 0.0,E4 0.0,E5 0.0,E6 0.0}
DECL FDAT FP47={TOOL_NO 1,BASE_NO 0,IPO_FRAME #BASE,POINT2[] " ",TQ_STATE FALSE}
DECL PDAT PPDAT129={VEL 100.0,ACC 100.0,APO_DIST 100.0,APO_MODE #CDIS}
DECL E6POS XP48={X 1834.22803,Y -6335.16309,Z 1712.83398,A -2.1284399,B 4.89814806,C 89.4969788,S 6,T 51,E1 -4829.7959,E2 0.0,E3 0.0,E4 0.0,E5 0.0,E6 0.0}
DECL FDAT FP48={TOOL_NO 1,BASE_NO 0,IPO_FRAME #BASE,POINT2[] " ",TQ_STATE FALSE}
DECL PDAT PPDAT130={VEL 100.0,ACC 100.0,APO_DIST 100.0,APO_MODE #CDIS}
DECL E6POS XP52={X 1834.22595,Y -6335.16797,Z 1712.80505,A -2.12861705,B 4.89925098,C 89.4980164,S 6,T 51,E1 -4829.7959,E2 0.0,E3 0.0,E4 0.0,E5 0.0,E6 0.0}
DECL FDAT FP52={TOOL_NO 1,BASE_NO 0,IPO_FRAME #BASE,POINT2[] " ",TQ_STATE FALSE}
DECL PDAT PPDAT134={VEL 100.0,ACC 100.0,APO_DIST 100.0,APO_MODE #CDIS}
DECL E6POS XP53={X 1407.51404,Y -6302.81787,Z 1750.83997,A -1.47880495,B 4.89941216,C 89.4990692,S 6,T 50,E1 -4829.7959,E2 0.0,E3 0.0,E4 0.0,E5 0.0,E6 0.0}
DECL FDAT FP53={TOOL_NO 1,BASE_NO 0,IPO_FRAME #BASE,POINT2[] " ",TQ_STATE FALSE}
DECL PDAT PPDAT135={VEL 100.0,ACC 100.0,APO_DIST 100.0,APO_MODE #CDIS}
DECL E6POS XP58={X 1733.22803,Y -6170.05322,Z 1660.64697,A -81.8373871,B -1.97206295,C -169.970795,S 2,T 35,E1 -4617.48682,E2 0.0,E3 0.0,E4 0.0,E5 0.0,E6 0.0}
DECL FDAT FP58={TOOL_NO 1,BASE_NO 0,IPO_FRAME #BASE,POINT2[] " ",TQ_STATE FALSE}
DECL PDAT PPDAT140={VEL 100.0,ACC 100.0,APO_DIST 100.0,APO_MODE #CDIS}
DECL E6POS XP59={X 1805.23706,Y -6520.43018,Z 1668.65601,A -81.8716125,B -2.00408602,C -156.326996,S 2,T 35,E1 -4617.48584,E2 0.0,E3 0.0,E4 0.0,E5 0.0,E6 0.0}
DECL FDAT FP59={TOOL_NO 1,BASE_NO 0,IPO_FRAME #BASE,POINT2[] " ",TQ_STATE FALSE}
DECL PDAT PPDAT141={VEL 100.0,ACC 100.0,APO_DIST 100.0,APO_MODE #CDIS}
DECL E6POS XP60={X 1764.02197,Y -6402.15576,Z 1650.85901,A -81.8596268,B -1.80446994,C -160.770798,S 2,T 35,E1 -4617.48682,E2 0.0,E3 0.0,E4 0.0,E5 0.0,E6 0.0}
DECL FDAT FP60={TOOL_NO 1,BASE_NO 0,IPO_FRAME #BASE,POINT2[] " ",TQ_STATE FALSE}
DECL PDAT PPDAT142={VEL 100.0,ACC 100.0,APO_DIST 100.0,APO_MODE #CDIS}
DECL PDAT PPDAT143={VEL 100.0,ACC 100.0,APO_DIST 100.0}
DECL E6POS XP62={X 956.073425,Y 883.9198,Z 30.4730206,A -97.7865372,B 10.2152596,C 10.5537996,S 6,T 19,E1 -4845.01709,E2 0.0,E3 0.0,E4 0.0,E5 0.0,E6 0.0}
DECL FDAT FP62={TOOL_NO 1,BASE_NO 2,IPO_FRAME #BASE,POINT2[] " ",TQ_STATE FALSE}
DECL PDAT PPDAT144={VEL 100.0,ACC 100.0,APO_DIST 100.0}
DECL PDAT PPDAT145={VEL 100.0,ACC 100.0,APO_DIST 100.0}
DECL PDAT PPDAT147={VEL 100.0,ACC 100.0,APO_DIST 100.0}
DECL PDAT PPDAT148={VEL 100.0,ACC 100.0,APO_DIST 100.0}
DECL PDAT PPDAT149={VEL 100.0,ACC 100.0,APO_DIST 100.0}
DECL PDAT PPDAT150={VEL 100.0,ACC 100.0,APO_DIST 100.0}
DECL PDAT PPDAT151={VEL 100.0,ACC 100.0,APO_DIST 100.0}
DECL E6POS XP71={X 954.767212,Y 883.147522,Z 26.7002602,A -93.6145172,B 14.0894003,C 6.16314602,S 6,T 19,E1 -4845.02002,E2 0.0,E3 0.0,E4 0.0,E5 0.0,E6 0.0}
DECL FDAT FP71={TOOL_NO 1,BASE_NO 2,IPO_FRAME #BASE,POINT2[] " ",TQ_STATE FALSE}
DECL PDAT PPDAT153={VEL 100.0,ACC 100.0,APO_DIST 100.0}
DECL E6POS XP73={X 2238.15088,Y 1920.05005,Z 256.481506,A -146.656494,B 11.9896402,C 89.91362,S 6,T 50,E1 -2992.02295,E2 0.0,E3 0.0,E4 0.0,E5 0.0,E6 0.0}
DECL FDAT FP73={TOOL_NO 1,BASE_NO 2,IPO_FRAME #BASE,POINT2[] " ",TQ_STATE FALSE}
DECL PDAT PPDAT155={VEL 100.0,ACC 100.0,APO_DIST 100.0}
DECL PDAT PPDAT157={VEL 100.0,ACC 100.0,APO_DIST 100.0}
DECL PDAT PPDAT158={VEL 100.0,ACC 100.0,APO_DIST 100.0}
DECL PDAT PPDAT159={VEL 100.0,ACC 100.0,APO_DIST 100.0}
DECL PDAT PPDAT160={VEL 100.0,ACC 100.0,APO_DIST 100.0}
DECL PDAT PPDAT161={VEL 100.0,ACC 100.0,APO_DIST 100.0}
DECL E6POS XP82={X 1305.98206,Y 902.312073,Z 35.7690697,A -168.313797,B -3.08961797,C -161.261703,S 2,T 35,E1 -4617.43311,E2 0.0,E3 0.0,E4 0.0,E5 0.0,E6 0.0}
DECL FDAT FP82={TOOL_NO 1,BASE_NO 2,IPO_FRAME #BASE,POINT2[] " ",TQ_STATE FALSE}
DECL PDAT PPDAT165={VEL 100.0,ACC 100.0,APO_DIST 100.0,APO_MODE #CDIS}
DECL E6POS XP83={X 1451.89697,Y 936.910583,Z 43.9505615,A -171.9422,B -1.59057796,C -155.522903,S 2,T 35,E1 -4617.45313,E2 0.0,E3 0.0,E4 0.0,E5 0.0,E6 0.0}
DECL FDAT FP83={TOOL_NO 1,BASE_NO 2,IPO_FRAME #BASE,POINT2[] " ",TQ_STATE FALSE}
DECL PDAT PPDAT166={VEL 100.0,ACC 100.0,APO_DIST 100.0,APO_MODE #CDIS}
DECL PDAT PPDAT167={VEL 100.0,ACC 100.0,APO_DIST 100.0}
DECL E6POS Xswp_60_0328={X 1442.66296,Y 881.827271,Z 43.2024117,A -156.052795,B -0.844046175,C -135.117996,S 2,T 35,E1 -4617.46484,E2 0.0,E3 0.0,E4 0.0,E5 0.0,E6 0.0}
DECL FDAT Fswp_60_0328={TOOL_NO 1,BASE_NO 2,IPO_FRAME #BASE,POINT2[] " ",TQ_STATE FALSE}
DECL E6POS Xswp_60_0324={X 1407.26404,Y 918.435974,Z 17.5869293,A -171.278397,B -1.13974595,C -144.781906,S 2,T 35,E1 -4617.40918,E2 0.0,E3 0.0,E4 0.0,E5 0.0,E6 0.0}
DECL FDAT Fswp_60_0324={TOOL_NO 1,BASE_NO 2,IPO_FRAME #BASE,POINT2[] " ",TQ_STATE FALSE}
DECL E6POS Xswp_60_0320={X 1355.86304,Y 916.699219,Z 15.1454897,A -171.2789,B -1.12584805,C -145.769897,S 2,T 35,E1 -4617.46484,E2 0.0,E3 0.0,E4 0.0,E5 0.0,E6 0.0}
DECL FDAT Fswp_60_0320={TOOL_NO 1,BASE_NO 2,IPO_FRAME #BASE,POINT2[] " ",TQ_STATE FALSE}
DECL E6POS XP84={X 452.798004,Y 879.223877,Z -176.399002,A -84.0717773,B 9.00781155,C -9.90915203,S 6,T 19,E1 -5459.74023,E2 0.0,E3 0.0,E4 0.0,E5 0.0,E6 0.0}
DECL FDAT FP84={TOOL_NO 1,BASE_NO 2,IPO_FRAME #BASE,POINT2[] " ",TQ_STATE FALSE}
DECL PDAT PPDAT168={VEL 100.0,ACC 100.0,APO_DIST 30.0,APO_MODE #CDIS}
DECL E6POS Xswp_60_0316={X 1315.01294,Y 874.13623,Z 40.566349,A -162.286697,B -5.82788897,C -156.920593,S 2,T 35,E1 -4617.43115,E2 0.0,E3 0.0,E4 0.0,E5 0.0,E6 0.0}
DECL FDAT Fswp_60_0316={TOOL_NO 1,BASE_NO 2,IPO_FRAME #BASE,POINT2[] " ",TQ_STATE FALSE}
ENDDAT
